PROGRAM ImpulseTest
VAR
	duration: LREAL := 2;
	torqueInput: REAL:= 0.05;
	torqueStarter : BOOL:= FALSE;
	state : INT := 10;	
	counter : LREAL := 0;	
	trial: INT := 5;
	delaytime: LREAL := 5000;
	counter1: LREAL := 0;
	counter3: LREAL :=0;
END_VAR

CASE state OF
10 :

	IF MAIN.dummy = 0 AND torqueStarter THEN
		state := 20;
	ELSIF MAIN.dummy = 1 AND torqueStarter THEN
		state := 30;
	END_IF
	
20 :
IF 	torqueStarter THEN
	counter := counter + MAIN.sampleTime;
	IF counter < duration THEN
			IF MAIN.opertionModeRead=10 THEN
				link.torqueX := REAL_TO_INT(torqueInput*(1000/2.37));	
			ELSIF MAIN.opertionModeRead=9 THEN				
				link.torqueOfsetX := LREAL_TO_INT(torqueInput*(1000/2.37));
			END_IF
	ELSE
		link.torqueX := 0;
		link.torqueOfsetX := 0;
		torqueStarter := FALSE;
		counter := 0;
		counter1:=0;			
		state := 60;
		
	END_IF
ELSE
	link.torqueX := 0;
	link.torqueOfsetX := 0;
END_IF
	
30 :
IF 	torqueStarter THEN
	counter := counter + MAIN.sampleTime;
	IF counter < duration THEN
			IF MAIN.opertionModeRead=10 THEN
				link.torqueY := REAL_TO_INT(torqueInput*(1000/2.37));	
			ELSIF MAIN.opertionModeRead=9 THEN				
				link.torqueOfsetY := LREAL_TO_INT(torqueInput*(1000/2.37));
			END_IF
	ELSE
		link.torqueY := 0;
		link.torqueOfsetY := 0;
		torqueStarter := FALSE;
		counter := 0;
		counter1:=0;		
		state := 60;
		
	END_IF
ELSE
	link.torqueY := 0;
	link.torqueOfsetY := 0;
END_IF

60 :
	counter1:=counter1+  MAIN.sampleTime;
	IF counter1<delaytime THEN
		torqueStarter:=FALSE;	
		counter := 0;
		
		ELSE
			counter3:=counter3+  1;	
			IF counter3 < trial THEN
				torqueStarter:=TRUE;		
				state :=10;
				counter := 0;
			ELSE
				torqueStarter:=FALSE;
				counter3 := 0;		
				state :=10;
				counter := 0;
				counter1 := 0;
				counter3 := 0;
		END_IF
	END_IF
END_CASE

END_PROGRAM

(* stored: Version 1.1.0.1, ProductVersion 3.1.4024.9
   POU ImpulseTest: Id {c390f270-7a3e-41da-ac54-2a0b3de05886}, SpecialFunc None *)
